(* IEC 61131-3 sources: MotionTestBenchMaster/Logical/12_MAU/1290_Logger/MAU_Logger, 2 files *)

(* ---- MAU_Logger.st ---- *)
PROGRAM _CYCLIC
	(* Software object logging *)
	swChg_0.refreshTime 		:= T#1m;
	swChg_0.logLevel			:= arEVENTLOG_SEVERITY_INFO;
	swChg_0.enable				:= TRUE;
	swChg_0();
END_PROGRAM

(* ---- Variables.var ---- *)
(*****************************************                  MACHINE SYNCHRONIZATION LOGGING             ***************************************************************************************************************)
VAR
	synchLog_0 : SynchLog;
END_VAR
(*****************************************                   UPS LOGGING                                                         ***************************************************************************************************************)
VAR
	upsIO : Sidel_UpsIo_typ;
	upsEvt : LogSupplyEvents;
END_VAR
(*****************************************                   SOFTWARE OBJECT LOGGING                               ***************************************************************************************************************)
VAR
	swChg_0 : SwChg;
	pippo :BOOL;
END_VAR
